PROGRAM MAIN_S1

VAR
	b110SyncState AT %I* :UINT ;
	b110State AT %I* :UINT;  
	EtherCATWCState23To49 AT %I* : BOOL; 
	EtherCATWCState50To76 AT %I* : BOOL; 
	AktiveSystem : BOOL := TRUE;
	bSwitch : BOOL := TRUE;
	nState: UINT;
	MoverState :ARRAY[1..GVL_MC.nNumMovers] OF UINT;
	nForCounter ,i: UINT;
	Velo : LREAL := 2000;
	//mover :ARRAY[1..nNumMovers] OF MC_PlanarMover;
	
	LocalSystemTime : FB_LocalSystemTime;
	
	fbTrackobject : FB_TrackObject;

	ipXlMover: 	I_XtsXlMover1;


	state : INT := -1;
	arrivedOTCID : OTCID;
	Start :BOOL;
	bAlldone : BOOL;
	
	

	test : otcid; 
	XPU_Number : UINT := 1; 	
	
	Short : BOOL := TRUE;
	
	XtsOutterLoopOid: OTCID ;	
	XtsShortcutOid: OTCID ;
	
	Init : BOOL ; 
	EndTrack : INT := E_TrackNum.MainEnd;
 	StartTrack : INT :=E_TrackNum.MainStart ;
	MoverNo : DINT;
	SystemReady: BOOL;
	IsDetectionOnStartupEnabled : BOOL := FALSE;
	
	MagnetValue AT%Q*: INT;
	bMagnetOn : BOOL;	
	Fault : BOOL;
	SwitchCurrent :lreal := 7;
	Switchcounter : DINT;
	FP_Counter : r_trig;
	

	aMoverTrack : ARRAY[1..GVL_Mc.nNumMovers] OF otcid;
	FirstMoverTrackPos : LREAL;
	MoverGap : LREAL;
	FTrigTrackCount : F_Trig;
	MoverNo1  : UDINT;
	gapStart: LREAL := 5600;
	gapLength: LREAL := 2000;
	moverInFront: UDINT;
	mover1FollowDist: LREAL;
	followSyncPos: LREAL;
	masterSyncPos: LREAL;
	masterPosAtSync: LREAL;
	followerPosAtSync: LREAL;
	endOfBigTrack : LREAL; 
     endOfSmallTrack : LREAL; 
     endOfMainTrack : LREAL; 
     followerToEndOfTrack: LREAL;
     leaderToEndofTrack: LREAL;
     distToMoverInFront: LREAL;
     vara: Tc3_Mc3PlanarMotion.PlanarObjectInfo;
  
     getList: BOOL;
     directMerge: BOOL;
     mergeNotPossible: BOOL;

	A : LREAL := 0.63;
	B : LREAL := 0.21;
	C : LREAL := 6;
	
	cmdFeedback: Tc3_XtsInterface.XtsCommandFeedback;
	BUFFER: BYTE;
	
	xReset AT %Q*: BOOL;
	xStart AT %Q*: BOOL;
	EtherCATFault: BOOL;
	syncFault: BOOL;

	
	haltDynamics : DynamicConstraint_PathXY;
	stMoverConfigSlow	: ST_MoverConfig;
	stMoverConfigNormal : ST_MoverConfig;
	stMoverConfigFast  : ST_MoverConfig;
	stMoverCfgAggressive : ST_MoverConfig;
	stMoverCfgHalt : ST_MoverConfig;
	MoverStopDone : BOOL;
	
	Fp_error : R_trig;
	
	ModuleState1 AT%I*: E_EcState;
	ModuleState2 AT%I*: E_EcState;
	ModuleState3 AT%I*: ARRAY[0..2] OF E_EcState;
	
	MessageTrigger : ARRAY[1..20] OF R_trig;
	
	
	TestPowerMat : BOOL := TRUE;
	StopTime : TIME := T#1S;
	StopTimer :ARRAY[1..nNumMovers] OF ton;
	StartTimer :ARRAY[1..nNumMovers] OF BOOL;
	SwitchParkPos : LREAL := 3500;
	trapError: BOOL;
	trapErrorID: UDINT;
	moverWithFault: UDINT;
	stepWithFault: INT;
	stopAndWait : ARRAY[1..nNumMovers] OF TON; 
	
	AllDone : BOOL;
	InitDone  :BOOL;
END_VAR


VAR_INPUT
	remoteState AT %I*: INT;
END_VAR


// =====================
// Initalize XTS Utility
GVL_MC.fbXtsEnvironment.Init(GVL_MC.cmdFeedback);
IF NOT GVL_MC.cmdFeedback.IsDone THEN
	RETURN;
END_IF


//=================== Check State of Modules===========================================
IF EtherCATWCState23To49 OR EtherCATWCState50To76 THEN 
	EtherCATFault := TRUE; 
END_IF
IF b110SyncState <> 1 THEN 
	syncFault := TRUE;  
END_IF

MessageTrigger[1](clk:=ModuleState1 <> 8 AND state> 0);
IF MessageTrigger[1].Q THEN
	ADSLOGSTR(msgCtrlMask:= ADSLOG_MSGTYPE_LOG , msgFmtStr:= 'Module Fault Line 1 %s' , strArg:= TO_STRING(ModuleState1));
END_IF

MessageTrigger[2](clk:=ModuleState2 <> 8 AND state> 0);
IF MessageTrigger[2].Q THEN
	ADSLOGSTR(msgCtrlMask:= ADSLOG_MSGTYPE_LOG , msgFmtStr:= 'Module Fault Line 2 %s ' , strArg:= TO_STRING(ModuleState2));
END_IF

MessageTrigger[3](clk:=ModuleState3[0] <> 8 AND state> 0);
IF MessageTrigger[3].Q THEN
	ADSLOGSTR(msgCtrlMask:= ADSLOG_MSGTYPE_LOG , msgFmtStr:= 'Module Fault Line 3 Default SyncUnit %s ' , strArg:= TO_STRING(ModuleState3[0]));
END_IF

MessageTrigger[4](clk:=ModuleState3[1] <> 8 AND state> 0);
IF MessageTrigger[4].Q THEN
	ADSLOGSTR(msgCtrlMask:= ADSLOG_MSGTYPE_LOG , msgFmtStr:= 'Module Fault Line 3 XtsTask SyncUnit %s ' , strArg:= TO_STRING(ModuleState3[1]));
END_IF

MessageTrigger[5](clk:=ModuleState3[2] <> 8 AND state> 0);
IF MessageTrigger[5].Q THEN
	ADSLOGSTR(msgCtrlMask:= ADSLOG_MSGTYPE_LOG , msgFmtStr:= 'Module Fault Line 3 PlcTask SyncUnit %s ' , strArg:= TO_STRING(ModuleState3[2]));
END_IF


//===========================================================================================

GVL_MC.ipXtsProcessingUnit :=  GVL_MC.fbXtsEnvironment.ProcessingUnit(XPU_Number,0);
FOR i := 1 TO GVL_MC.nNumMovers DO 	
	
	IF NOT InitDone  THEN
		ipXlMover  :=  GVL_MC.fbXtsEnvironment.ProcessingUnit(XPU_Number, 0).XlMover(i, 0);
		AllDone := AllDone AND GVL_MC.fbMover[i].Init(ipXlMover, GVL_MC.ipXtsProcessingUnit); 
	END_IF
	InitDone := alldone;
	
	Fp_error(clk := GVL_MC.fbMover[i].P_PlanarMover.Error AND GVL_MC.fbMover[i].XtsXlMover.GetIsActive(0) AND state = 100);
	IF Fp_error.Q THEN
		state := 140;
		Fault := TRUE;

		ADSLOGSTR(msgCtrlMask:= ADSLOG_MSGTYPE_LOG , msgFmtStr:= 'Mover %s Faulted ' , strArg:= INT_TO_STRING(i));
	ELSE
		Fault := FALSE;
	END_IF
	
	
	GVL_MC.Feedback[i].Update();
	GVL_MC.fbMover[i].CycleUpdate();
	GVL_MC.iMover[i] := GVL_MC.fbMover[i];
	GVL_MC.fbMover[i].P_Dynamics.SetValuesVADJ(Velo, 4000, 4000, 16000);
	GVL_MC.fbMover[i].P_MoveOnTrackOptions.gap := 900;
	GVL_MC.fbMover[i].P_MoveOnTrackOptions.direction := MC_Direction.mcDirectionPositive;
	GVL_MC.fbMover[i].P_MoveOnTrackOptions.gapMode := MC_GAP_MODE_ON_TRACK.Fast1D;
	
	GVL_DataExchange.aMoverInfos[i] :=  GVL_MC.fbMover[i].P_MoverInfos;
END_FOR	

fbTrackobject(TrackID:= GVL_mc.aMcTracks[E_TrackNum.big].MCTOPLC_STD.TrackOID,iMover:= gvl_mc.iMover ); 
fbTrackobject.CyclicUpdate();

FOR i := 1 TO GVL_MC.nNumTracks DO 
	GVL_MC.aMcTracks[i].Update();
	GVL_MC.TrackFeedback[i].Update();
END_FOR	

IF NOT Init THEN
	Init := TRUE;
END_IF




GVL_DataExchange.Dynamics.v := Velo;

IF state < 99 AND xReset THEN 
	IF State = 1 THEN 
		xReset := FALSE; 
	END_IF 
	state := 0; 
END_IF
IF state = 99 AND xStart AND remoteState  = 99 THEN   
	state := 100;  
END_IF

CASE state OF
	0: 
		
		FOR i := 1 TO GVL_MC.nNumTracks DO  
			GVL_MC.aMcTracks[i].Enable(GVL_MC.TrackFeedback[i]);
			state := 1;
		END_FOR
		
	1: 	
		bAlldone := TRUE;
		FOR i := 1 TO GVL_MC.nNumTracks DO  
			bAlldone := bAlldone AND GVL_MC.aMcTracks[i].MCTOPLC_STD.State = MC_PLANAR_STATE.Enabled ;
		END_FOR

 		IF bAlldone THEN
			state := 2;
		END_IF

	2:	
	
		FOR i := 1+GVL_MC.nNumActiveMovers TO GVL_MC.nNumMovers DO  
			GVL_MC.fbMover[i].XlProcessingUnit.XlMover(i,0).SetStartupTrackPosition(0.2,0);	
			GVL_MC.fbMover[i].XlProcessingUnit.XlMover(i,0).SetIsVirtualFeedbackEnabled(1,0);
			GVL_MC.fbMover[i].XlProcessingUnit.XlMover(i,0).TriggerArrive(0);
		END_FOR
		IF  GVL_MC.nNumActiveMovers > 0 THEN
			FOR i :=1  TO GVL_MC.nNumActiveMovers DO 	
				GVL_MC.fbMover[i].XlProcessingUnit.XlMover(i,0).SetIsVirtualFeedbackEnabled(0,0);
			END_FOR 
		END_IF			
		state := 3;
		
	3:
		FOR i := 1 TO GVL_MC.fbXtsEnvironment.ProcessingUnit(1, 0).XlPartCount() DO
			 GVL_MC.fbXtsEnvironment.ProcessingUnit(1, 0).XlPart(i, 0).TriggerReset(0);
		END_FOR
		
		state := 5;
		
	5: 

		
		IF AktiveSystem THEN
			state := 10;
		ELSE
			state := 100;
		END_IF	

	10:
		FOR i := 1 TO GVL_MC.nNumActiveMovers DO
			GVL_MC.fbMover[i].P_PlanarMover.Reset(0);			
		END_FOR
		state := 11; 
	11:
		FOR i := 1 TO GVL_MC.nNumActiveMovers DO
			GVL_MC.fbMover[i].P_PlanarMover.Enable(0);		
		END_FOR
		state := 15;	
	15:
		bAlldone := TRUE;
		FOR i := 1 TO GVL_MC.nNumActiveMovers DO  
			bAlldone := bAlldone AND GVL_MC.fbMover[i].P_PlanarMover.MCTOPLC.STD.State = MC_PLANAR_STATE.Enabled ;	
		END_FOR
		
		IF bAlldone THEN
			state := 18;
		END_IF
	18: 
	
		FOR i := 1 TO GVL_MC.nNumActiveMovers DO  
			GVL_MC.fbMover[i].JoinNearestTrack(aMcTracks,nNumTracks);	
		END_FOR
		state := 20;
	
	20:
		bAlldone := TRUE;
		FOR i := 1 TO GVL_MC.nNumActiveMovers DO  
			bAlldone := bAlldone AND GVL_MC.fbMover[i].fbPlanarMover.MCTOPLC.STD.CommandMode = MC_PLANAR_MOVER_COMMAND_MODE.OnTrack  ;	
			MoverState[i] := 10;
			
		END_FOR

		IF bAlldone THEN
			state := 99;
			Fault := FALSE;
		END_IF
		
	99:
	 	IF GVL_MC.nNumActiveMovers = 0 THEN
			state := 100;
		END_IF
		
	100: 
		arrivedOTCID := GVL_MC.EnterSystem.PopFirstMoverInQueue();
		IF arrivedOTCID <> 0 THEN
			FOR i := 1  TO GVL_MC.nNumMovers DO
				IF GVL_MC.fbMover[i].P_MoverOTCID = arrivedOTCID THEN
					MoverState[i] := 0;
				END_IF
			END_FOR
		END_IF
	
		FOR i := 1 TO GVL_MC.nNumMovers DO 
			
			IF MoverNo1 <> 0 AND_THEN GVL_MC.fbMover[MoverNo1].P_PlanarMover.MCTOPLC.SETONTRACK.TrackOID =  GVL_MC.aMcTracks[E_TrackNum.Big].MCTOPLC_STD.TrackOID THEN
				Short := FALSE;
			END_IF	
		
			CASE MoverState[i] OF 
			0:		 
				IF  bSwitch AND GVL_MC.fbMover[i].P_PlanarMover.MCTOPLC.SETONTRACK.TrackOID = GVL_MC.aMcTracks[E_TrackNum.MainStart].MCTOPLC_STD.TrackOID    THEN
					IF NOT short   THEN
						GVL_MC.fbMover[i].MoveOnTrack(GVL_MC.aMcTracks[E_TrackNum.Small], SwitchParkPos(* GVL_MC.aMcTracks[E_TrackNum.Small].GetLength()/2*), GVL_MC.defaultGap);
						MoverNo1 := i;
						Short := TRUE;
						MoverState[i] := 6;
					ELSE
						GVL_MC.fbMover[i].MoveOnTrack(GVL_MC.aMcTracks[E_TrackNum.Big],(GVL_MC.aMcTracks[E_TrackNum.Big].GetLength()-12000), GVL_MC.defaultGap);			
						MoverState[i] := 10;
					END_IF
				ELSIF NOT bSwitch AND  GVL_MC.fbMover[i].P_PlanarMover.MCTOPLC.SETONTRACK.TrackOID = GVL_MC.aMcTracks[E_TrackNum.MainStart].MCTOPLC_STD.TrackOID THEN
					GVL_MC.fbMover[i].MoveOnTrack(GVL_MC.aMcTracks[EndTrack],GVL_MC.aMcTracks[EndTrack].GetLength()-450, GVL_MC.defaultGap);
					MoverState[i] := 12;				
				END_IF
			4:
				IF fbMover[i].P_PlanarFeedback.Error AND NOT trapError THEN //trap the error once.   
						trapError := fbMover[i].P_PlanarFeedback.Error; 
						trapErrorID := fbMover[i].P_PlanarFeedback.ErrorId;
						stepWithFault := 4;
 						moverWithFault := i; 
					END_IF
					IF fbMover[i].P_PlanarFeedback.Done THEN 
						MoverState[i] := 5; //50;
						stopAndWait[i](IN:=TRUE, PT:=StopTime); 
					END_IF 	
			5:
				stopAndWait[i](); 
					IF stopAndWait[i].Q  OR NOT TestPowerMat THEN // send the mover to a sync Position 2.6m before the end of the track 
						stopAndWait[i](IN:=FALSE); 							
						MoverState[i] := 6; 
					END_IF 	
				
			6:
               
                fbTrackobject.findMergePosition(
                   mergeSyncCommandPos := gapStart , 
                   spaceToMerge := gapLength, 
                   nMoverToFollow => moverInFront, 
                   mergeWithoutFollow => directMerge, 
                   mergeNotPossible => mergeNotPossible); 
								
                IF (directMerge OR moverInFront <> 0) AND NOT mergeNotPossible THEN
                                MoverState[i] := 7;
                END_IF 
			7:  //merge with gap zero
					//issue commmand to sync 
					IF  directMerge THEN 
						GVL_MC.fbMover[i].P_Dynamics.SetValuesVADJ(stMoverConfigNormal.velo,stMoverConfigNormal.Accel,stMoverConfigNormal.Decel,stMoverConfigNormal.Jerk);
						fbMover[i].MoveOnTrack(track:= GVL_Mc.aMCTracks[E_TrackNum.MainEnd], targetPos:= GVL_Mc.aMCtracks[E_TrackNum.Mainend].GetLength()-500, gap:= GVL_MC.defaultGap);

						MoverState[i] := 10; 
					ELSIF moverInFront <>0 THEN 
						fbMover[i].P_Dynamics.SetValuesVADJ(stMoverConfigNormal.velo,stMoverConfigNormal.Accel,stMoverConfigNormal.Decel,stMoverConfigNormal.Jerk);
						masterSyncPos := GVL_Mc.aMCTracks[E_TrackNum.Big].GetLength()-2500;
						masterPosAtSync := Mover[moverInFront].MoverPos; 
						followSyncPos := GVL_Mc.aMCTracks[E_TrackNum.Small].GetLength()- GVL_MC.defaultGap -2500;
						followerPosAtSync :=Mover[nForCounter].MoverPos; 
						fbMover[i].SyncToOtherMover( 
							masterSyncPos := masterSyncPos,
							masterTrack := GVL_Mc.aMCTracks[E_TrackNum.Big],
							followerSyncPos := followSyncPos,
							followerTrack := GVL_Mc.aMCTracks[e_TrackNum.Small],
							PlanarMoverToFollow := fbMover[moverInFront].P_PlanarMover,
							velo:= stMoverConfigNormal.velo);
							MoverState[i] := 8; 
						// reduce the gap of the leading mover 
						fbMover[moverInFront].MoveOnTrack(track:= GVL_Mc.aMcTracks[E_TrackNum.Big], targetPos:= GVL_Mc.aMcTracks[E_TrackNum.Big].GetLength()-500, gap:= 0);

					END_IF 
			
  			
                  
  			8: // wait for in Sync 
                  IF Gvl_mc.fbMover[i].P_SyncFeedback.Active AND  gvl_mc.MOver[moverInFront].TrackID =  GVL_Mc.aMCTracks[E_TrackNum.Big].MCTOPLC_STD.TrackOID THEN // actively syncing calculate distance from mover 
                  		
						followerToEndOfTrack := endOfSmallTrack - gvl_mc.Mover[i].MoverPos; 
                  		leaderToEndofTrack := endOfBigTrack - gvl_mc.Mover[moverInFront].MoverPos; 
                  		distToMoverInFront := followerToEndOfTrack - leaderToEndofTrack; 
						
                  ELSE 
                 		followerToEndOfTrack := 0; 
                 		leaderToEndofTrack := 0; 
                 		distToMoverInFront := 0;
                  END_IF
				  
               	IF fbMover[nForCounter].P_SyncFeedback.inSync OR  MOver[nForCounter].TrackID =  GVL_Mc.aMCTracks[E_TrackNum.MainEnd].MCTOPLC_STD.TrackOID THEN 
						MoverState[i] := 10;
						Short :=FALSE;
				ELSIF	fbMover[nForCounter].P_SyncFeedback.Error THEN
						MoverState[i] := 6;
				END_IF 

			10:

				IF SystemReady AND (  GVL_MC.fbMover[i].P_PlanarMover.MCTOPLC.SETONTRACK.SetPos > 500 AND GVL_MC.fbMover[i].P_PlanarMover.MCTOPLC.SETONTRACK.TrackOID <>  GVL_MC.aMcTracks[StartTrack].MCTOPLC_STD.TrackOID) THEN
					GVL_MC.fbMover[i].MoveOnTrack(GVL_MC.aMcTracks[EndTrack], GVL_MC.aMcTracks[EndTrack].GetLength()- 200, GVL_MC.defaultGap);
					MoverState[i] := 12;
				END_IF
		
			12: 
				//500mm after that the boundary change commmand is issued 
				IF GVL_MC.fbMover[i].P_PlanarMover.MCTOPLC.SETONTRACK.SetPos > GVL_MC.aMcTracks[E_TrackNum.MainEnd].GetLength() - 2300 AND // 2300
				(GVL_MC.fbMover[i].P_PlanarMover.MCTOPLC.SETONTRACK.TrackOID = GVL_MC.aMcTracks[E_TrackNum.MainEnd].MCTOPLC_STD.TrackOID)  THEN 
					GVL_MC.fbMover[i].LeaveSystemAt(GVL_MC.ExitSystem, GVL_MC.defaultGap); 
					MoverState[i] := 15; 
				END_IF
				
			15:
			 	IF GVL_MC.fbMover[i].XlProcessingUnit.XlMover(i,0).GetIsVirtualFeedbackEnabled(0) AND //In some cases the planar mover gots an error, we have to evaluate why
					GVL_MC.fbMover[i].P_PlanarMover.Error THEN
					GVL_MC.fbMover[i].P_PlanarMover.Reset(0);
					MoverState[i] := 16; 
				END_IF
				
			16: 
				GVL_MC.fbMover[i].P_PlanarMover.Disable(0);
				MoverState[i] := 17; 
		
			END_CASE
		END_FOR	
		
		140:
			FOR i := 1 TO GVL_MC.nNumMovers DO  
				GVL_MC.fbMover[i].P_PlanarMover.Halt(GVL_MC.Feedback[i], haltDynamics);
			END_FOR	
			
				state := 145;
			
		145:
			bAllDone := TRUE;
				FOR i := 1 TO GVL_MC.nNumMovers DO  
				IF NOT(GVL_MC.Feedback[i].Done OR GVL_MC.Feedback[i].Error) THEN
					bAllDone := FALSE;
					EXIT;
				END_IF
			END_FOR
			
			IF bAllDone THEN
				state := 150;
			END_IF
		
		//Disable
		150:
			MoverStopDone := TRUE;
			FOR i := 1 TO GVL_MC.nNumMovers DO  
					GVL_MC.fbMover[i].P_PlanarMover.Disable(GVL_MC.Feedback[i]);
			END_FOR
				
			state := 0;
		
		
	
END_CASE

//bMagnetOn := FALSE;
FOR nForCounter:=1 TO GVL_MC.nNumMovers DO
	
//	IF  GVL_MC.fbMover[nForCounter].XtsXlMover.GetPositionInfo_trackObjectId(0) = GVL_mc.XtsShortcutOid AND (IsBetween(GVL_MC.fbMover[nForCounter].XtsXlMover.GetPositionInfo_trackPosition(0), gvl_mc.fMagnetEntry - (Velo*0.06), gvl_mc.fMagnetExit(*- Velo*0.04*))) THEN
//		bMagnetOn := TRUE;
//	END_IF
END_FOR


		SwitchCurrent := ((A*(((Velo/1000)*(Velo/1000))))+(B*(Velo/1000))+C);
IF bMagnetOn AND NOT Fault THEN

	MagnetValue := TO_INT(SwitchCurrent*1310);
ELSE
 	MagnetValue := 0;
END_IF

FP_Counter(clk:=bMagnetOn);

IF FP_Counter.Q THEN
	Switchcounter := Switchcounter+1;

END_IF

//distanceMonitoring of Mover 1 when on the big track 
IF GVL_MC.Mover[1].TrackID = GVL_Mc.aMcTracks[E_TrackNum.MainStart].MCTOPLC_STD.TrackOID THEN //calculate out how far it is to the mover in front 
	IF GVL_MC.Mover[moverInFront].MoverPos -  GVL_Mc.Mover[1].MoverPos > 10 THEN 
		mover1FollowDist := GVL_Mc.Mover[moverInFront].MoverPos -  GVL_Mc.Mover[1].MoverPos;
	END_IF   
END_IF

END_PROGRAM

(* stored: Version 1.1.0.1, ProductVersion 3.1.4026.11
   POU MAIN_S1: Id {1e7add0e-820a-414b-96de-5fe81886ac49}, SpecialFunc None *)
